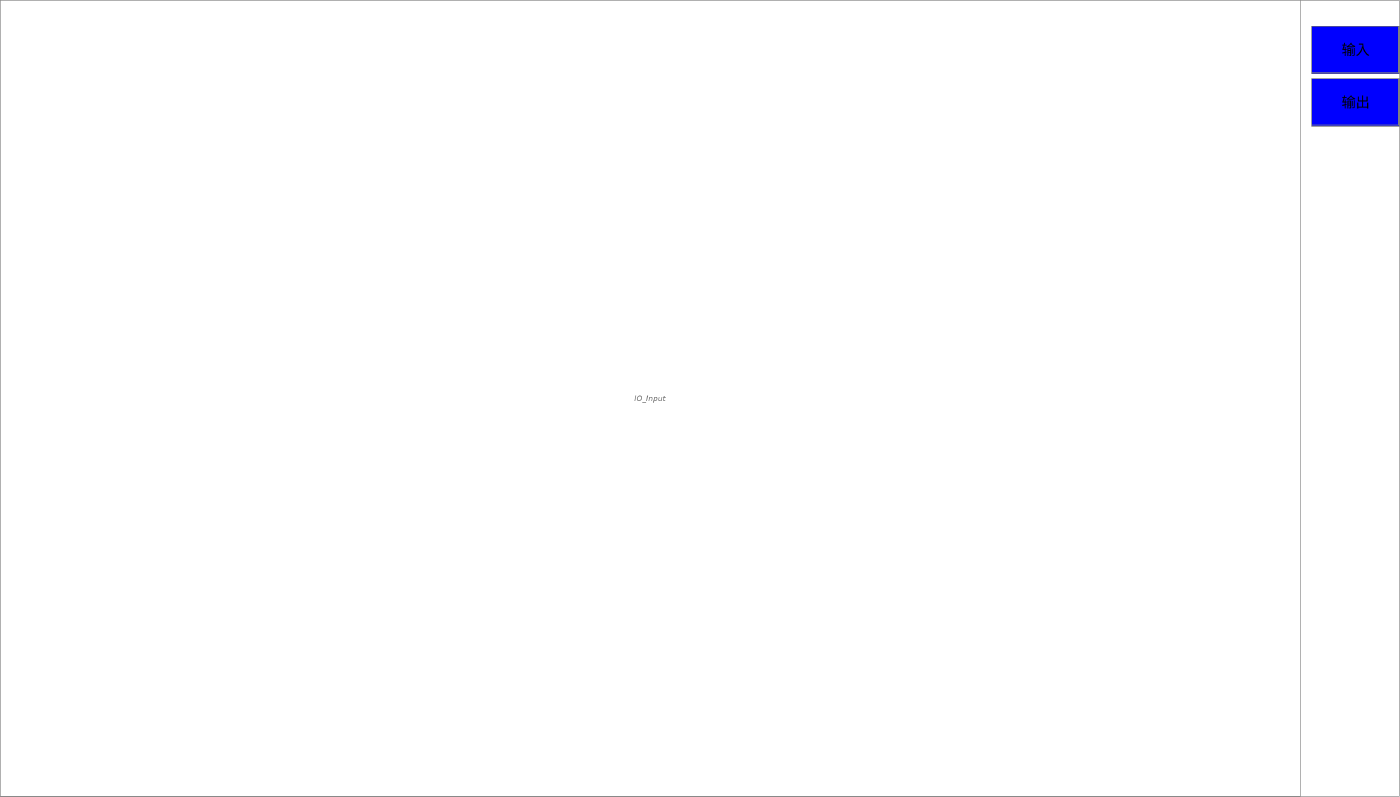
VISUALIZATION IO  // 1895x1080
    Frame (0,0 1760x1080)
        shows IO_Input()
        shows IO_Output()
        shows Auto_test_1()
    Button (1775,35 120x65), "输入"
        OnMouseClick: FrameSelectionChange Selection=SelectedFrame=1d4c33e9-a5b9-451d-bf86-00d28fadf65b, GlobSel=AssignType=Directly, SelType=Locally
    Button (1775,106 120x65), "输出"
        OnMouseClick: FrameSelectionChange Selection=SelectedFrame=1d4c33e9-a5b9-451d-bf86-00d28fadf65b, Selection=1, GlobSel=AssignType=Directly, SelType=Locally
END_VISUALIZATION

(* stored: Version 1.1.0.1, ProductVersion 3.1.4024.4
   Visu IO: Id {609c1598-65c2-4cd9-9d27-4211d33d5d3d} *)
